VAR_GLOBAL
	hmiHeaderInstance	:	FB_HMIHeader;
	hmiHeaderInterface	:	HMIHeader;	
	hmiOperatingmodeInterface	:	HMIInterfaceOperatingMode;
	
	hmiAdsCommunicationInterfaceInstance	:	FB_ADSCommunicationStatus;
	hmiAdsCommunicationInterface	:	ADSCommunicationInterface;
	
	hmiMachineSectionInterface	:	MachineSectionHMIInterface;
	
	hmiEmitterInstances	:	ARRAY[0..1] OF STRING := [
														'Zufuehrband',
														'SubParts'
													];
	hmiConveyorInstances	:	ARRAY[0..1] OF STRING := [
															'Foerderband 6',
															'Zufuehrung'
														 ];
	hmiElevatorInstances	:	ARRAY[0..1] OF STRING := [
															'Einlauf',
															'Hochregallager'
														];
	hmiStackerCraneInstances	:	ARRAY[0..1] OF STRING := [
															'Einlagerung',
															'Auslagerung'
														 ];		
	hmiRFIDInstances	:	ARRAY[0..2] OF STRING := [
															'Einlagerung',
															'Zufuehrung',
															'Warehouse-Infeed'
														 ];	
	hmiPositingBarInstances	:	ARRAY[0..2] OF STRING := [
															'Blau laden',
															'Gruen laden',
															'Grau laden'
														 ];										 
	hmiPickPlaceInstances	:	ARRAY[0..2] OF STRING := [
															'Einlagerung',
															'Zufuehrung',
															'Warehouse-Infeed'
														 ];	
	hmiRemoverInstances	:	ARRAY[0..1] OF STRING := [
														'Zufuehrband',
														'SubParts'
													];
END_VAR

(* stored: Version 1.1.0.1
   GVL HMI: Id {42b8ab01-74f8-4d3b-9b14-9c080998c4d7} *)
